// TIA Portal project "enkoder_asenkron motor_kontrolu" (V18)

(* hardware
DEVICE "S7-1200 station_1"  S7-1200 Station
   slot 0: "Rack_0"  S7-1200 Rack  Rack  V1.0
   slot 1: "PLC_1"  CPU 1214C DC/DC/DC  6ES7 214-1AG40-0XB0  V4.6
*)

// ===== PLC "PLC_1"  CPU 1214C DC/DC/DC =====

VAR_GLOBAL   // PLC tag table "Default tag table"
   "Tag_1" AT %M20.0 : Bool;
   "Tag_2" AT %MD60 : DWord;
   "HSC5_ADRESI" AT %ID1016 : DWord;
   "HSC5_ATAMA" AT %MD30 : DWord;
   "START" AT %I0.0 : Bool;
   "START ÇIKIŞ" AT %Q0.0 : Bool;
   "YÖN" AT %Q0.1 : Bool;
   "Tag_3" AT %M70.0 : Bool;
   "Tag_4" AT %I0.1 : Bool;
   "HIZ BİLGİSİ" AT %Q0.3 : Bool;
   "Tag_5" AT %M50.0 : Bool;
   "ACİL STOP" AT %I0.7 : Bool;
END_VAR

// folder: System blocks/Program resources

DATA_BLOCK "T1"   // DB2
{ S7_Optimized_Access := 'TRUE' }
AUTHOR : Simatic
FAMILY : IEC
NAME : IEC_TMR
VERSION : 1.0
// stored: InstanceOfName IEC_TIMER
"IEC_TIMER"
BEGIN
END_DATA_BLOCK

// folder: (top level)

ORGANIZATION_BLOCK "Main"   // OB1, LAD, ProgramCycle
TITLE = "Main Program Sweep (Cycle)"
{ S7_Optimized_Access := 'TRUE' }
VERSION : 0.1
   VAR_INPUT
      Initial_Call : Bool;   // Initial call of this OB
      Remanence : Bool;   // =True, if remanent data are available
   END_VAR
   VAR_TEMP   // added for the SCL form of the ladder/FBD networks
      _w1 : Bool;
   END_VAR
BEGIN

REGION Network 1
   // enkoder abz fazlı
   // 1 turda 500 pulse
   // motor 20 tur attığında dursun =10000pulse
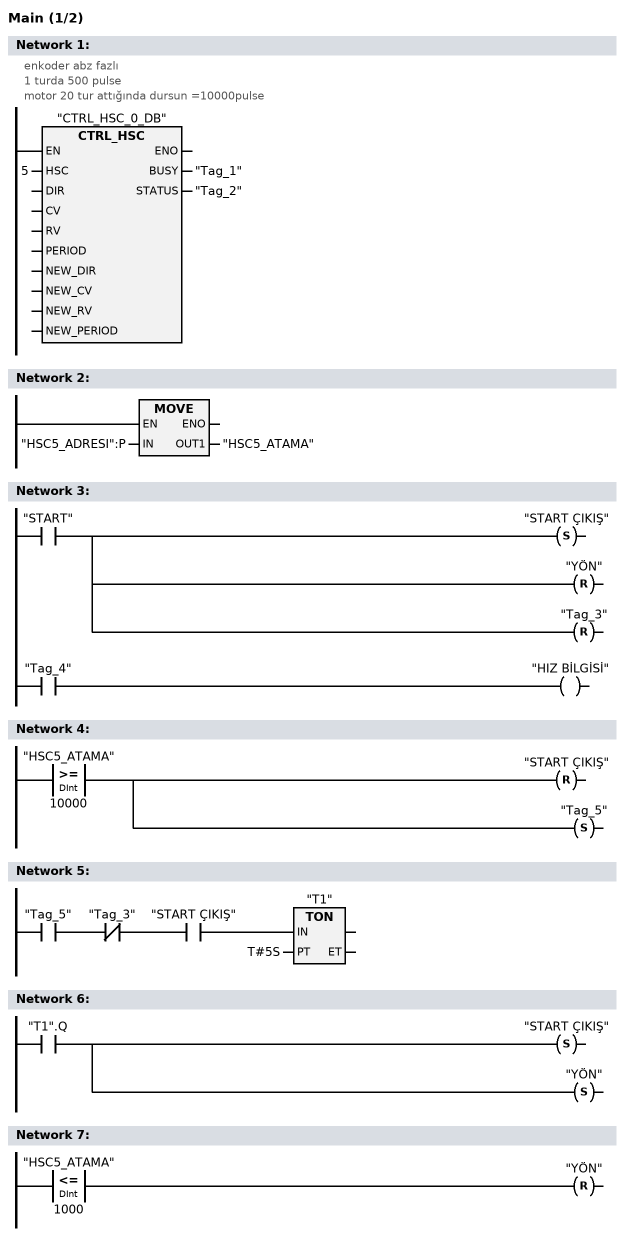
   "CTRL_HSC_0_DB"(HSC := 5, BUSY => "Tag_1", STATUS => "Tag_2");   // CTRL_HSC
END_REGION

REGION Network 2
   RUNG wire#powerrail
      Move(in := "HSC5_ADRESI":P, out1 => "HSC5_ATAMA")
   END_RUNG
   // the same network as SCL:
   "HSC5_ATAMA" := "HSC5_ADRESI":P;
END_REGION

REGION Network 3
   RUNG wire#powerrail
      Contact( "START" )
      wire#w1
      S_Coil( "START ÇIKIŞ" )
   END_RUNG
   RUNG wire#w1
      R_Coil( "YÖN" )
   END_RUNG
   RUNG wire#w1
      R_Coil( "Tag_3" )
   END_RUNG
   RUNG wire#powerrail
      Contact( "Tag_4" )
      Coil( "HIZ BİLGİSİ" )
   END_RUNG
   // the same network as SCL:
   IF "START" THEN
       "START ÇIKIŞ" := TRUE;
       "YÖN" := FALSE;
       "Tag_3" := FALSE;
   END_IF;
   "HIZ BİLGİSİ" := "Tag_4";
END_REGION

REGION Network 4
   RUNG wire#powerrail
      { S7_Templates := "SrcType := DInt" } GE_Contact(in1 := "HSC5_ATAMA", in2 := 10000)
      wire#w1
      R_Coil( "START ÇIKIŞ" )
   END_RUNG
   RUNG wire#w1
      S_Coil( "Tag_5" )
   END_RUNG
   // the same network as SCL:
   IF "HSC5_ATAMA" >= 10000 THEN
       "START ÇIKIŞ" := FALSE;
       "Tag_5" := TRUE;
   END_IF;
END_REGION

REGION Network 5
   "T1".TON(IN := "Tag_5" AND NOT "Tag_3" AND "START ÇIKIŞ", PT := T#5S);
END_REGION

REGION Network 6
   RUNG wire#powerrail
      Contact( "T1".Q )
      wire#w1
      S_Coil( "START ÇIKIŞ" )
   END_RUNG
   RUNG wire#w1
      S_Coil( "YÖN" )
   END_RUNG
   // the same network as SCL:
   IF "T1".Q THEN
       "START ÇIKIŞ" := TRUE;
       "YÖN" := TRUE;
   END_IF;
END_REGION

REGION Network 7
   RUNG wire#powerrail
      { S7_Templates := "SrcType := DInt" } LE_Contact(in1 := "HSC5_ATAMA", in2 := 1000)
      R_Coil( "YÖN" )
   END_RUNG
   // the same network as SCL:
   IF "HSC5_ATAMA" <= 1000 THEN "YÖN" := FALSE; END_IF;
END_REGION

REGION Network 8
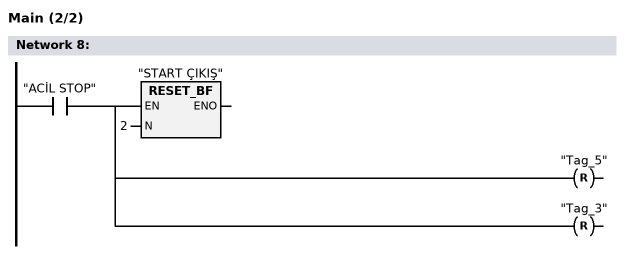
   // no SCL statement known for RBitfield: written as a call
   #_w1 := "ACİL STOP";
   IF #_w1 THEN
       RESET_BF(operand := "START ÇIKIŞ", n := 2);
       "Tag_5" := FALSE;
       "Tag_3" := FALSE;
   END_IF;
END_REGION
END_ORGANIZATION_BLOCK